FUNCTION_BLOCK FB_Values
VAR_INPUT
END_VAR
VAR_OUTPUT
END_VAR
VAR

//Function Blocks	
	fbSineFast:GEN;
	fbCosineFast:GEN;
	fbTriangleFast:GEN;
	fbSineSlow:GEN;
	fbCosineSlow:GEN;
	fbTriangleSlow:GEN;
	
//FB Outputs
	iSineFast: INT;
	iCosineFast: INT;
	iTriangleFast: INT;
	iSineSlow: INT;
	iCosineSlow: INT;
	iTriangleSlow: INT;
	
END_VAR

(*
-signal generator

*)

//sine fast
fbSineFast(
	MODE:=SINE , 
	BASE:=TRUE , 
	PERIOD:=T#500MS , 
	CYCLES:= , 
	AMPLITUDE:=100 , 
	RESET:= , 
	OUT=>iSineFast );
	
//cosine
fbCoSineFast(
	MODE:=COSINE , 
	BASE:=TRUE , 
	PERIOD:=T#600MS , 
	CYCLES:= , 
	AMPLITUDE:=100 , 
	RESET:= , 
	OUT=>iCosineFast );

//triangular
fbTriangleFast(
	MODE:=TRIANGLE , 
	BASE:=TRUE , 
	PERIOD:=T#700MS , 
	CYCLES:= , 
	AMPLITUDE:=200 , 
	RESET:= , 
	OUT=>iTriangleFast );


//sine
fbSineSlow(
	MODE:=SINE , 
	BASE:=TRUE , 
	PERIOD:=T#5S , 
	CYCLES:= , 
	AMPLITUDE:=100 , 
	RESET:= , 
	OUT=>iSineSlow );
	
//cosine
fbCoSineSlow(
	MODE:=COSINE , 
	BASE:=TRUE , 
	PERIOD:=T#6S , 
	CYCLES:= , 
	AMPLITUDE:=100 , 
	RESET:= , 
	OUT=>iCosineSlow );

//triangular
fbTriangleSlow(
	MODE:=TRIANGLE , 
	BASE:=TRUE , 
	PERIOD:=T#7S , 
	CYCLES:= , 
	AMPLITUDE:=200 , 
	RESET:= , 
	OUT=>iTriangleSlow );

PROPERTY CosineFast : REAL
GET
CosineFast:=TO_REAL(iCosineFast);
END_GET
END_PROPERTY

PROPERTY CosineSlow : REAL
GET
CosineSlow:=TO_REAL(iCosineSlow);
END_GET
END_PROPERTY

PROPERTY SineFast : REAL
GET
SineFast:=TO_REAL(iSineFast);
END_GET
END_PROPERTY

PROPERTY SineSlow : REAL
GET
SineSlow:=TO_REAL(iSineFast);
END_GET
END_PROPERTY

PROPERTY TriangleFast : REAL
GET
TriangleFast:=TO_REAL(iTriangleFast);
END_GET
END_PROPERTY

PROPERTY TriangleSlow : REAL
GET
TriangleSlow:=TO_REAL(iTriangleSlow);
END_GET
END_PROPERTY

END_FUNCTION_BLOCK

(* stored: Version 1.1.0.1, ProductVersion 3.1.4024.12
   POU FB_Values: Id {0deb296a-535b-41f4-ae81-dd6782819b37}, SpecialFunc None
   Property CosineFast: Id {45d31ca9-f4d8-417d-a9fd-bb2021eacf8d}
   Get Get: Id {b6ae8773-e956-431f-a78d-a68971aabb84}
   Property CosineSlow: Id {a9ffcf1f-8127-4bf6-8d59-afb12b3c3b6b}
   Get Get: Id {4f837de8-f215-45f7-880c-7eb889986798}
   Property SineFast: Id {3418f0cc-bf0f-4bbf-bcaa-3af1a5d7d96f}
   Get Get: Id {09a65b4e-70a0-46e6-8e5c-088053ad08d7}
   Property SineSlow: Id {607627a6-ee98-4692-9f2c-c4367c0e3e8f}
   Get Get: Id {e6432fee-33a8-40de-9758-351a59874280}
   Property TriangleFast: Id {39382217-9318-4601-a5ab-536bdfa91965}
   Get Get: Id {31b48053-0934-454a-97eb-8167c798e0a5}
   Property TriangleSlow: Id {fc6336e7-2a62-440b-9ded-32d08b7ab683}
   Get Get: Id {2ad2021c-f05a-49dd-b3b4-c5bf35b1738d} *)
